(* IEC 61131-3 sources: cybercode_codesys_lib/src/basic/mechanism, 4 files *)

(* ---- E_FeedbackState.st ---- *)
TYPE E_FeedbackState  :
(
    Inactive                   := 0,   // Обратная связь неактивна (норма при остановке)
    Active                     := 1,   // Обратная связь активна (норма при работе)
    Error_NoFeedback           := 2,   // Нет обратной связи при наличии питания
    Error_UnexpectedFeedback   := 3    // Обратная связь есть при отсутствии питания
);
END_TYPE

(* ---- FB_AbstractMechanism.st ---- *)
FUNCTION_BLOCK ABSTRACT FB_AbstractMechanism
VAR_INPUT
END_VAR
VAR_OUTPUT
END_VAR
VAR
END_VAR

METHOD SetPower
VAR_INPUT
    x : BOOL;
END_VAR
    _xPower := x;
END_METHOD

METHOD GetPower : BOOL
VAR_INPUT
END_VAR
GetPower := _xPower;
END_METHOD

METHOD ABSTRACT Start
VAR_INPUT
END_VAR
END_METHOD

METHOD ABSTRACT Stop
VAR_INPUT
END_VAR
END_METHOD

END_FUNCTION_BLOCK

(* ---- FB_Mechanism.st ---- *)
FUNCTION_BLOCK FB_Mechanism EXTENDS FB_AbstractMechanism
VAR_INPUT
END_VAR
VAR_OUTPUT
END_VAR
VAR
END_VAR

METHOD Start
VAR_INPUT
END_VAR
    SetPower(TRUE);
END_METHOD

METHOD Stop
VAR_INPUT
END_VAR
    SetPower(FALSE);
END_METHOD

END_FUNCTION_BLOCK

(* ---- FB_MechanismWithFeedback.st ---- *)
FUNCTION_BLOCK FB_MechanismWithFeedback EXTENDS FB_Mechanism
VAR_INPUT
	ixFeedback : BOOL;
END_VAR
VAR_OUTPUT
END_VAR
VAR
	_uFeedbackState : E_StateFeedback;
END_VAR

    UpdateState();

METHOD GetFeedbackWithoutPower : BOOL
VAR_INPUT
END_VAR
    GetFeedbackWithoutPower := _uFeedbackState = E_StateFeedback.Error_UnexpectedFeedback;
END_METHOD

METHOD GetPowerAndFeedback : BOOL
VAR_INPUT
END_VAR
    GetPowerAndFeedback := _uFeedbackState = E_StateFeedback.Active;
END_METHOD

METHOD GetPowerWithoutFeedback : BOOL
VAR_INPUT
END_VAR
    GetPowerWithoutFeedback := _uFeedbackState = E_StateFeedback.Error_NoFeedback;
END_METHOD

METHOD GetState : UINT
VAR_INPUT
END_VAR
    GetState := _uFeedbackState;
END_METHOD

METHOD PROTECTED UpdateState
VAR_INPUT
END_VAR
    IF NOT GetPower() AND NOT ixFeedback THEN _uFeedbackState := E_StateFeedback.Inactive; END_IF; 				// 0
    IF GetPower() AND ixFeedback THEN _uFeedbackState := E_StateFeedback.Active; END_IF; 						// 1
    IF GetPower() AND NOT ixFeedback THEN _uFeedbackState := E_StateFeedback.Error_NoFeedback; END_IF;			// 2
    IF NOT GetPower() AND ixFeedback THEN _uFeedbackState := E_StateFeedback.Error_UnexpectedFeedback; END_IF;	// 3
END_METHOD

END_FUNCTION_BLOCK
